///////////
// Structure For Battery Racks. Main Operating Data to be saved ( ex: OPC ) .  
//////////
TYPE RackString_KP :
STRUCT
	
		MesData		: RackString ;

		
     	
	
		

		
		
		
		
		
		
		
	
END_STRUCT
END_TYPE

(* stored: Version 1.1.0.1, ProductVersion 3.1.4024.12
   DUT RackString_KP: Id {0301049b-59db-4d95-8b96-2ff155a80608} *)
